TYPE ST_HMIDigInputs :
STRUCT
END_STRUCT
END_TYPE

(* stored: Version 1.1.0.1, ProductVersion 3.1.4024.12
   DUT ST_HMIDigInputs: Id {856a834f-0a9d-4c88-8f4f-88b3463c6d1b} *)
